TYPE "MatCounterWng"
VERSION : 0.1
// Block: MatCounterWng
   STRUCT
      EncoderNotValid : Bool;
      EncoderPosNotValid : Bool;
      PresetRunning : Bool;
   END_STRUCT;

END_TYPE
